# EPICS SNL sequencer program: viocs/bo_rf/bo_rfApp/src/rf_sp_init.stt
program rf_sp_init

int event_proc;
assign event_proc to "EVENT-BO-05D:RF-Cav:SP-INIT.PROC";

ss ss1 {
    state init {
        when (delay(1.0)) {
            event_proc = 1;
            pvPut(event_proc);
        } exit
    }
}
